// TIA Portal V20 export
// export: Created 2025-12-01T14:57:44.3031575Z, ExportSetting None, DisplayName Totally Integrated Automation Portal, DisplayVersion V20 Update 3, DisplayName TIA Portal Openness, DisplayVersion V20 Update 3, DisplayName TIA Portal Version Control Interface, DisplayVersion V20 Update 3, DisplayName STEP 7 Professional, DisplayVersion V20 Update 3, DisplayName STEP 7 Safety, DisplayVersion V20 Update 2, DisplayName WinCC Basic/Comfort/Advanced, DisplayVersion V20 Update 3, DisplayName WinCC Professional, DisplayVersion V20 Update 3, DisplayName WinCC Unified, DisplayVersion V20 Update 3
FUNCTION "FC532_Estado_Ocupacion" : Void   // FC532, STL
{ S7_Optimized_Access := 'FALSE' }
AUTHOR : ROUTER
NAME : 20130631
VERSION : 3.1
// stored: AutoNumber false
   VAR_INPUT
      NumeroMesa : UInt;   // Numero de Mesa
      EstadoMesaVacia : Bool;   // Vacia=1
      MesaDeJDT02 : Bool;
   END_VAR
   VAR_IN_OUT
      MemEstadoOcupa : Byte;
   END_VAR
   VAR_TEMP
      DBEventos : Word;   // Numero del DB de Eventos
      NumBytes : UInt;   // Numero de Bytes existentes en el DB de Eventos
      PunteroEventos : DWord;   // Puntero al DB de Eventos
      ValorTMP : UDInt;
      OffsetTMP : UInt;
      NumDBEventos : UInt;
      MaxBytes : UInt;
   END_VAR
BEGIN

NETWORK
TITLE = 
// ---------------------------------------------------------------------
// --- Mirar si estamos activos para mandar el estado de la mesa

      SET;
      A     "DB902_Estado_ZonaMesa".EstadoMesas[#NumeroMesa].Marcha_CBx;  //#Estado_Zona_Mesa.Marcha_CBx
      JC    Continua;

      L     0;
      T     #MemEstadoOcupa;

      JU    Fin_funcion;



NETWORK
TITLE = Acciones
// ---------------------------------------------------------------------
// --- Mirar el Estado de Ocupacion de la Mesa (Si ha Cambiado)

Continua:SET;  // Mirar si ha cambiado de Estado
      A     #EstadoMesaVacia;  // Estado diferente
      A(;
      O(;
      L     #MemEstadoOcupa;
      L     2;
      ==I;
      );
      O(;
      L     #MemEstadoOcupa;
      L     0;
      ==I;
      );
      );
      JC    Emitir_estado;

      SET;
      AN    #EstadoMesaVacia;
      A(;
      O(;
      L     #MemEstadoOcupa;
      L     1;
      ==I;
      );
      O(;
      L     #MemEstadoOcupa;
      L     0;
      ==I;
      );
      );
      JC    Emitir_estado;

      JU    Fin_funcion;  // No ha Cambiado de Estado


NETWORK
TITLE = Evento de Estado de Ocupacion de la Mesa
// ---------------------------------------------------------------------
// ---
// ---
// ---   Pasos a Seguir para el Formateo del Evento
// ---
// ---   * Mirar si hay sitio para generar el nuevo evento
// ---       * Inicializo NumBytes y Puntero al DB de Eventos Generados
// ---       * Calcula el tamaño de bytes que hay en el DB de Eventos Generados
// ---       * Comprobar si hay sitio para un evento más
// ---   *  Formatear el Evento
// ---
// ---
// ---------------------------------------------------------------------


// ---------------------------------------------------------------------
// --- Mirar si hay sitio para generar un evento más

Emitir_estado:SET;
      L     "JDT1_NDB_EventosEmi";
      T     #DBEventos;
      T     #NumDBEventos;
      L     "JDT1_MaxBytes";
      T     #MaxBytes;

// ---------------------------------------------------------------------
/// Inicio --> Pertenece al JDT 02

      AN    #MesaDeJDT02;
      JC    No_es_JdT02;

      L     "JDT2_NDB_EventosEmi";
      T     #DBEventos;
      T     #NumDBEventos;
      L     "JDT2_MaxBytes";
      T     #MaxBytes;

No_es_JdT02:NOP   0;

/// Final --> Pertenece al JDT 02
// ---------------------------------------------------------------------


      L     0;
      T     #NumBytes;  // Inicializo el numero de Bytes
      T     #PunteroEventos;  // Inicializo el puntero de Eventos Generados


Buscar_hueco:SET;
      OPN   DB [#DBEventos];  // Calcula el tamaño de bytes que hay en el DB
      L     DBB [#PunteroEventos];
      L     0;
      ==I;
      JC    Valida_hueco;  // Buscamos el final del DB = 0

      OPN   DB [#DBEventos];
      L     DBB [#PunteroEventos];
      L     ' ';
      ==I;
      JC    Valida_hueco;  // Buscamos el final del DB = ' '

      L     #PunteroEventos;  // Incremento de P#1.0
      L     P#1.0;
      +D;
      T     #PunteroEventos;

      JU    Buscar_hueco;  // Continuar con el siguiente posicion


Valida_hueco:SET;
      L     #PunteroEventos;  // Sacamos el NumBytes Escritos
      SRD   3;
      T     #NumBytes;

      L     #NumBytes;  // Miramos si hay sitio
      L     #MaxBytes;  // Max. que se pueden emitir, parametro
      >I;
      JC    Fin_funcion;  // No se pueden generar más eventos

// ---------------------------------------------------------------------
// --- Formatear el evento de Estado de Ocupacion de la Mesa

      L     #PunteroEventos;
      LAR2;  // Puntero al DB de Eventos Generados

      TAR2;  // Mirar si es el primer evento de la lista
      L     0;
      ==I;
      JC    Primer_evento;  // Es el primero

      OPN   DB [#DBEventos];
      L     ',';  // Separador entre eventos ','
      T     DBB [AR2, P#0.0];
      +AR2  P#1.0;


Primer_evento:SET;
      OPN   DB [#DBEventos];  // DB de Eventos Generados (A Emitir)
      L     '{';  // Inicio de Evento '{'
      T     DBB [AR2, P#0.0];
      +AR2  P#1.0;

      L     'DIDA';  // --- Evento 'DIDA'
      T     DBD [AR2, P#0.0];
      +AR2  P#4.0;

      OPN   DB [#DBEventos];
      L     '[';  // --- Evento - Atributo Tipo '[TIPO]'
      T     DBB [AR2, P#0.0];
      L     'TIPO';
      T     DBD [AR2, P#1.0];
      L     ']';
      T     DBB [AR2, P#5.0];
      +AR2  P#6.0;

      OPN   DB [#DBEventos];
      L     'MESA';  // Tipo Llave 'MESA'
      T     DBD [AR2, P#0.0];
      +AR2  P#4.0;

      L     '[';  // --- Evento - Atributo Numero de Mesa '[NUME]'
      T     DBB [AR2, P#0.0];
      L     'NUME';
      T     DBD [AR2, P#1.0];
      L     ']';
      T     DBB [AR2, P#5.0];
      +AR2  P#6.0;

      L     "CTE_OffsetMesa";
      L     #NumeroMesa;  // Numero de la Llave
      +I;
      T     #ValorTMP;

// --- Convertir Valor a ASCII

      TAR2;
      SRD   3;
      T     #NumBytes;  // Miro que offset tiene la String

      CALL  "FC893_Obtener_StringDelAtributo"
      ( DB_String := #NumDBEventos,
        OffsetIni := #NumBytes,
        Valor     := #ValorTMP,
        OffsetFin := #OffsetTMP
      );  // Llamo a ObtenerStrinAtributo

      L     #OffsetTMP;
      SLD   3;
      LAR2;  // Recupero que offset tiene la String

// --- Ya esta convertido el Valor a ASCII

      OPN   DB [#DBEventos];
      L     '[';  // --- Evento - Atributo de Estado '[FULL]'
      T     DBB [AR2, P#0.0];
      L     'FULL';
      T     DBD [AR2, P#1.0];
      L     ']';
      T     DBB [AR2, P#5.0];
      +AR2  P#6.0;

      L     'VACI';
      SET;
      A     #EstadoMesaVacia;
      JC    _EST;

      L     'LLEN';

_EST: OPN   DB [#DBEventos];
      T     DBD [AR2, P#0.0];
      +AR2  P#4.0;

      OPN   DB [#DBEventos];  // DB de Eventos Generados (A Emitir)
      L     '}';  // --- Fin de Evento '}'
      T     DBB [AR2, P#0.0];
      +AR2  P#1.0;

// ---------------------------------------------------------------------
// --- Final del Evento

      SET;
      A     #EstadoMesaVacia;
      JCN   VACI;
      L     DINT#1;
      T     #MemEstadoOcupa;

VACI: SET;
      AN    #EstadoMesaVacia;
      JCN   Fin_funcion;

      L     DINT#2;
      T     #MemEstadoOcupa;

      JU    Fin_funcion;  //Final del Formateo del Elento


NETWORK
TITLE = Final de la Funcion
// ---------------------------------------------------------------------
// --- Final de la Funcion

Fin_funcion:NOP   0;

END_FUNCTION
